// TIA Portal V20 export
TYPE "Tank"
   STRUCT
      isTankFull : Bool;
      tankLevel : Int;
      isEmpty : Bool;
      "type" : Bool;
   END_STRUCT;
END_TYPE
